// Mitsubishi GX Works2 project: Sequence2   PLC: Q03UDV

PROGRAM MAIN
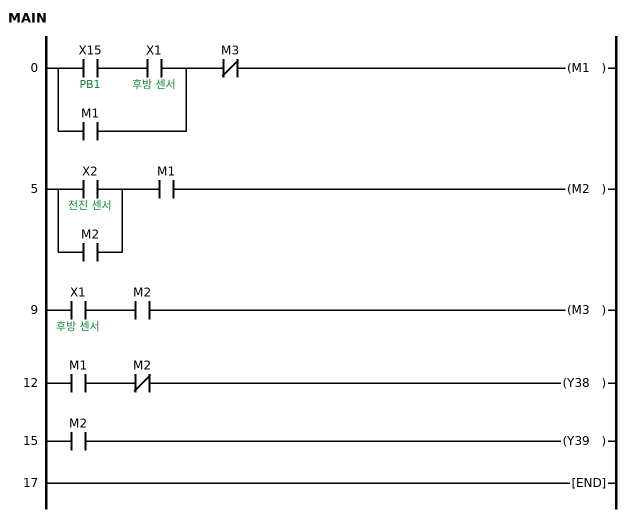
0     LD      X15  ; PB1
      AND     X1  ; 후방 센서
      OR      M1
      ANI     M3
      OUT     M1
5     LD      X2  ; 전진 센서
      OR      M2
      AND     M1
      OUT     M2
9     LD      X1  ; 후방 센서
      AND     M2
      OUT     M3
12    LD      M1
      ANI     M2
      OUT     Y38
15    LD      M2
      OUT     Y39
17    END
END_PROGRAM
